(* IEC 61131-3 sources: plc_generation_empirical_study/datasets/_archive/native_profile_v6_20260811/tasks/C02_H01_fault_lockout_reset, 2 files *)

(* ---- interface.st ---- *)
FUNCTION_BLOCK C02_H01_fault_lockout_reset
VAR_INPUT
    Start : BOOL;
    Stop : BOOL;
    Fault : BOOL;
    Reset : BOOL;
    Permit : BOOL;
END_VAR
VAR_OUTPUT
    Running : BOOL;
    LockedOut : BOOL;
END_VAR
END_FUNCTION_BLOCK

(* ---- reference.st ---- *)
FUNCTION_BLOCK C02_H01_fault_lockout_reset
VAR_INPUT
    Start : BOOL;
    Stop : BOOL;
    Fault : BOOL;
    Reset : BOOL;
    Permit : BOOL;
END_VAR
VAR_OUTPUT
    Running : BOOL;
    LockedOut : BOOL;
END_VAR

IF Fault THEN
    LockedOut := TRUE;
    Running := FALSE;
ELSIF Reset AND (NOT Start) THEN
    LockedOut := FALSE;
END_IF;

IF LockedOut OR Stop OR (NOT Permit) THEN
    Running := FALSE;
ELSIF Start THEN
    Running := TRUE;
END_IF;

END_FUNCTION_BLOCK
